(* IEC 61131-3 sources: factoryforge/examples/openplc/tank-level-control, 1 file *)

(* ---- tank_level_control.st ---- *)
(* ------------------------------------------------------------------------
   FactoryForge starter -- Tank level control (scene tank-level-control)
   OpenPLC Runtime v3, IEC 61131-3 Structured Text, over Modbus TCP.
   Generated by tools/gen_starters.py from the scene's tag set; see README.md
   beside this file. Write your program in section 2 below.

   THE TASK
     Hold the tank at the level the panel's pot asks for, using the fill
     and drain valves. Outflow follows Torricelli, so the process gain
     changes with level: a controller tuned at the top overshoots at the
     bottom.

   DONE WHEN
     The level settles within a few percent of the setpoint and holds
     there, and it still settles after you move the pot to a different
     level. A seized valve (tank.fault) keeps its opening while your
     command reads zero.

   HOW IT IS WIRED
     FactoryForge is the Modbus slave; OpenPLC is the master and polls it.
     mbconfig.cfg beside this file is that Slave Device. The addresses
     below are the ones the sidecar serves for this scene when it is
     started AFTER the scene is open, in the folder FactoryForge was
     extracted to:

       .\factoryforge-sidecar connect --driver modbus-tcp -o port 5502

     (./factoryforge-sidecar on Linux.)
     It prints its address map on startup; that map is the authority, and
     the table below must match it line for line. Change scene and the
     sidecar keeps every address it has handed out and puts new tags above
     them -- restart it after changing scene.

     OpenPLC numbers each block it polls from 100: slave coil n is
     %QX(100 + n/8).(n mod 8), slave input register n is %IW(100 + n).

     An INT or REAL tag is 32 bits and takes TWO registers, high word
     first. Section 1 rebuilds the inputs and section 3 splits the outputs;
     your program works with the plain DINT and REAL variables.

     In the sidecar's order (block, then address; addresses are decimal):

     MODBUS   REGS  OPENPLC                TAG
     0x0      1     %QX100.0               panel.green
     0x1      1     %QX100.1               panel.red
     0x2      1     %QX100.2               tower.green
     0x3      1     %QX100.3               tower.red
     0x4      1     %QX100.4               tower.yellow
     1x0      1     %IX100.0               panel.estop
     1x1      1     %IX100.1               panel.reset
     1x2      1     %IX100.2               panel.start
     1x3      1     %IX100.3               panel.stop
     1x4      1     %IX100.4               tank.fault
     4x0      2     %QW100 + %QW101        level_readout.value
     4x2      2     %QW102 + %QW103        tank.drain
     4x4      2     %QW104 + %QW105        tank.fill
     3x0      2     %IW100 + %IW101        panel.setpoint
     3x2      2     %IW102 + %IW103        tank.level
   ------------------------------------------------------------------------ *)

(* A REAL arrives the same way: IEEE-754 single precision, high word first.
   OpenPLC's DWORD_TO_REAL cannot rebuild it -- it converts the NUMBER, so
   16#3F800000 becomes 1065353216.0 rather than 1.0 -- so this takes the
   sign, exponent and mantissa apart by hand. Exact for every normal value;
   zero and the tiny subnormals (below 1.2E-38) come back as 0.0. *)
FUNCTION FF_WORDS_TO_REAL : REAL
  VAR_INPUT
    HI : WORD;
    LO : WORD;
  END_VAR
  VAR
    Exponent : INT;
    Value    : REAL;
  END_VAR
  Exponent := WORD_TO_INT(SHR(IN := HI, N := 7) AND 16#00FF);
  IF Exponent = 0 OR Exponent = 255 THEN
    Value := 0.0;
  ELSE
    Value := 1.0 + DWORD_TO_REAL(SHL(IN := WORD_TO_DWORD(HI AND 16#007F), N := 16)
                                 OR WORD_TO_DWORD(LO)) / 8388608.0;
    Exponent := Exponent - 127;
    WHILE Exponent > 0 DO
      Value := Value * 2.0;
      Exponent := Exponent - 1;
    END_WHILE;
    WHILE Exponent < 0 DO
      Value := Value / 2.0;
      Exponent := Exponent + 1;
    END_WHILE;
    IF (HI AND 16#8000) <> 0 THEN
      Value := -Value;
    END_IF;
  END_IF;
  FF_WORDS_TO_REAL := Value;
END_FUNCTION

(* The other direction: a REAL as the 32 bits IEEE-754 gives it, for
   splitting into two registers. REAL_TO_DWORD cannot do this either (it
   rounds the number). Exact for every normal value; anything smaller than
   1.2E-38 is sent as zero. *)
FUNCTION FF_REAL_TO_DWORD : DWORD
  VAR_INPUT
    IN : REAL;
  END_VAR
  VAR
    Magnitude : REAL;
    Exponent  : INT;
    Sign      : DWORD;
  END_VAR
  Sign := 0;
  Magnitude := IN;
  IF Magnitude < 0.0 THEN
    Sign := 16#80000000;
    Magnitude := -Magnitude;
  END_IF;
  Exponent := 127;
  WHILE Magnitude >= 2.0 AND Exponent < 254 DO
    Magnitude := Magnitude / 2.0;
    Exponent := Exponent + 1;
  END_WHILE;
  WHILE Magnitude < 1.0 AND Exponent > 1 DO
    Magnitude := Magnitude * 2.0;
    Exponent := Exponent - 1;
  END_WHILE;
  IF Magnitude < 1.0 THEN
    FF_REAL_TO_DWORD := Sign;
  ELSIF Magnitude >= 2.0 THEN
    FF_REAL_TO_DWORD := Sign OR 16#7F7FFFFF;
  ELSE
    FF_REAL_TO_DWORD := Sign
                        OR SHL(IN := INT_TO_DWORD(Exponent), N := 23)
                        OR REAL_TO_DWORD((Magnitude - 1.0) * 8388608.0);
  END_IF;
END_FUNCTION

PROGRAM tank_level_control
  VAR
    (* --- PLC writes: coils --------------------------------------------- *)
    PanelGreen  AT %QX100.0  : BOOL;  (* panel.green  0x0   green lamp on the panel *)
    PanelRed    AT %QX100.1  : BOOL;  (* panel.red    0x1   red lamp on the panel *)
    TowerGreen  AT %QX100.2  : BOOL;  (* tower.green  0x2   tower lamp, green *)
    TowerRed    AT %QX100.3  : BOOL;  (* tower.red    0x3   tower lamp, red *)
    TowerYellow AT %QX100.4  : BOOL;  (* tower.yellow 0x4   tower lamp, yellow *)
    (* --- PLC writes: holding registers, two per value ------------------ *)
    LevelReadoutValueHi AT %QW100    : WORD;  (* level_readout.value 4x0   high word of LevelReadoutValue *)
    LevelReadoutValueLo AT %QW101    : WORD;  (* level_readout.value 4x1   low word of LevelReadoutValue *)
    TankDrainHi         AT %QW102    : WORD;  (* tank.drain          4x2   high word of TankDrain *)
    TankDrainLo         AT %QW103    : WORD;  (* tank.drain          4x3   low word of TankDrain *)
    TankFillHi          AT %QW104    : WORD;  (* tank.fill           4x4   high word of TankFill *)
    TankFillLo          AT %QW105    : WORD;  (* tank.fill           4x5   low word of TankFill *)
    (* --- PLC reads: discrete inputs ------------------------------------ *)
    PanelEstop AT %IX100.0  : BOOL;  (* panel.estop 1x0   E-stop, normally closed: TRUE = healthy, FALSE = pressed; stays pressed until pulled out *)
    PanelReset AT %IX100.1  : BOOL;  (* panel.reset 1x1   Reset button, momentary: a short pulse per press *)
    PanelStart AT %IX100.2  : BOOL;  (* panel.start 1x2   Start button, momentary: a short pulse per press -- latch it *)
    PanelStop  AT %IX100.3  : BOOL;  (* panel.stop  1x3   Stop button, momentary: a short pulse per press *)
    TankFault  AT %IX100.4  : BOOL;  (* tank.fault  1x4   valve fault: TRUE = a valve has seized and holds its opening, whatever you command *)
    (* --- PLC reads: input registers, two per value --------------------- *)
    PanelSetpointHi AT %IW100    : WORD;  (* panel.setpoint 3x0   high word of PanelSetpoint *)
    PanelSetpointLo AT %IW101    : WORD;  (* panel.setpoint 3x1   low word of PanelSetpoint *)
    TankLevelHi     AT %IW102    : WORD;  (* tank.level     3x2   high word of TankLevel *)
    TankLevelLo     AT %IW103    : WORD;  (* tank.level     3x3   low word of TankLevel *)
  END_VAR

  (* A second VAR block, and not for tidiness: matiec will not mix located
     and unlocated declarations in one. Your own variables go here too. *)
  VAR
    (* --- PLC reads, in engineering units ---------------------------------- *)
    PanelSetpoint     : REAL;  (* panel.setpoint the operator's pot, 0..100 % (starts at 70) *)
    TankLevel         : REAL;  (* tank.level     tank level, % of capacity *)
    (* --- PLC writes, in engineering units ---------------------------------- *)
    LevelReadoutValue : DINT;  (* level_readout.value number shown on the display (%) *)
    TankDrain         : REAL;  (* tank.drain          drain valve opening, 0..100 % *)
    TankFill          : REAL;  (* tank.fill           fill valve opening, 0..100 % *)
    Raw32 : DWORD;  (* scratch for splitting a 32-bit output *)
  END_VAR

  (* ===== 1. Inputs: rebuild each 32-bit value from its two registers ===== *)
  PanelSetpoint := FF_WORDS_TO_REAL(HI := PanelSetpointHi, LO := PanelSetpointLo);
  TankLevel := FF_WORDS_TO_REAL(HI := TankLevelHi, LO := TankLevelLo);

  (* ===== 2. Your program ================================================
     The task is at the top of this file and in the scene's Task panel.
     Every signal above can be used by name here: the bits directly, the
     32-bit values through PanelSetpoint, TankLevel, LevelReadoutValue,
     TankDrain, TankFill. *)

  (* ===== 3. Outputs: split each 32-bit value into its two registers ===== *)
  Raw32 := DINT_TO_DWORD(LevelReadoutValue);
  LevelReadoutValueHi := DWORD_TO_WORD(SHR(IN := Raw32, N := 16));
  LevelReadoutValueLo := DWORD_TO_WORD(Raw32);
  Raw32 := FF_REAL_TO_DWORD(TankDrain);
  TankDrainHi := DWORD_TO_WORD(SHR(IN := Raw32, N := 16));
  TankDrainLo := DWORD_TO_WORD(Raw32);
  Raw32 := FF_REAL_TO_DWORD(TankFill);
  TankFillHi := DWORD_TO_WORD(SHR(IN := Raw32, N := 16));
  TankFillLo := DWORD_TO_WORD(Raw32);

END_PROGRAM

CONFIGURATION Config0

  RESOURCE Res0 ON PLC
    (* 20 ms, as in examples/openplc/Sorting.st: every scan spent waiting
       comes out of the scene's timing margins. *)
    TASK Main(INTERVAL := T#20ms, PRIORITY := 0);
    PROGRAM Inst0 WITH Main : tank_level_control;
  END_RESOURCE

END_CONFIGURATION
